FUNCTION_BLOCK Path1d EXTENDS ZCore.Object IMPLEMENTS IPathQuery, IPathQuery2, IPathQuery3, ZCore.IUnmanagedObject
VAR
  _owner : REFERENCE TO Unit;
  _fromPosition, _toPosition : LREAL;
  _direction : INT;
  _halfWidth, _safetyMargin : LREAL;
  _regions : POINTER TO ZApplication.IRegion;
  _regionEnd : INT;
  
  _maxRegions : DINT := 5;
  _regionIndicesBuffer1 : ARRAY[0..5] OF INT;
  _regionIndicesBuffer2 : ARRAY[0..5] OF INT;  
  _regionLockIndices : ZCore.RingBufferInt(_maxRegions, ADR(_regionIndicesBuffer1));
  _regionUnlockIndices : ZCore.RingBufferInt(_maxRegions, ADR(_regionIndicesBuffer2));
END_VAR

METHOD CheckAndLock : BOOL;
VAR_INPUT
  pos : LREAL;
END_VAR
VAR_INST
  i : DINT;
  region : ZApplication.IRegion;
  corner1WithMargin, corner2WithMargin : Vector4;
END_VAR
IF _regionLockIndices.Empty
THEN
  CheckAndLock := TRUE;
  RETURN;
END_IF

region := _regions[_regionLockIndices.ItemAt(0)];
CheckAndLock := 
  region.IntersectsIntervalX(pos - _halfWidth - _safetyMargin, pos + _halfWidth + _safetyMargin) AND_THEN
  region.TryLock(_owner);
  
IF CheckAndLock
THEN
  _regionUnlockIndices.Append(_regionLockIndices.ItemAt(0));
END_IF
END_METHOD

PROPERTY CurrentEdge : LREAL
GET
IF _regionLockIndices.Empty
THEN
  CurrentEdge := _toPosition;
  RETURN;
END_IF

IF _direction < 0
THEN
  CurrentEdge := _regions[_regionLockIndices.ItemAt(0)].Corner2.X + _halfWidth;
ELSE
  CurrentEdge := _regions[_regionLockIndices.ItemAt(0)].Corner1.X - _halfWidth;
END_IF
END_GET
END_PROPERTY

METHOD Cyclic
VAR_INST
  i : DINT;
  region : ZApplication.IRegion;
  priority : INT;
  priorityIndex : DINT;
  waiting : BOOL;
END_VAR
IF NOT Busy
THEN
  RETURN;
END_IF

IF _regionLockIndices.Empty
THEN
  SetBusy(FALSE);  
  RETURN;
END_IF

priority := 10000;
FOR i := 0 TO _regionLockIndices.Size - 1
DO
  region := _regions[_regionLockIndices.ItemAt(i)];
  IF priority > region.Priority
  THEN
    priorityIndex := i;
    priority := region.Priority;
  END_IF
END_FOR

waiting := FALSE;
FOR i := priorityIndex TO _regionLockIndices.Size - 1
DO
  region := _regions[_regionLockIndices.ItemAt(i)];
  IF NOT region.TryLock(_owner)
  THEN
    waiting := TRUE;
  END_IF
END_FOR

SetBusy(waiting);

// We can't move so free up resources
IF Busy
THEN
  FOR i := 0 TO _regionLockIndices.Size - 1
  DO
    region := _regions[_regionLockIndices.ItemAt(i)];
    region.Unlock(_owner);
  END_FOR
END_IF
END_METHOD

//FB_Init is always available implicitly and it is used primarily for initialization.
//The return value is not evaluated. For a specific influence, you can also declare the
//methods explicitly and provide additional code there with the standard initialization
//code. You can evaluate the return value.
METHOD FB_Init: BOOL
VAR_INPUT
    bInitRetains: BOOL; // TRUE: the retain variables are initialized (reset warm / reset cold)
    bInCopyCode: BOOL;  // TRUE: the instance will be copied to the copy code afterward (online change)   
END_VAR
SetIdle();
END_METHOD

METHOD FromPosition : IPathQuery2
VAR_INPUT
  pos : LREAL;
END_VAR
_fromPosition := pos;

FromPosition := THIS^;
END_METHOD

METHOD IncrementRegion
VAR_INST
  intervalMin : LREAL;
  intervalMax : LREAL;
  i : INT;
  
  corner1, corner2 : Vector4;
END_VAR
IF NOT _regionLockIndices.Empty
THEN
  _regionLockIndices.PopFirstItem();
END_IF
END_METHOD

PROPERTY RegionsToPass : DINT
GET
RegionsToPass := _regionLockIndices.Size;
END_GET
END_PROPERTY

METHOD ReserveAsync
VAR_INPUT
  unit : REFERENCE TO Unit;
END_VAR
VAR_INST
  intervalMin : LREAL;
  intervalMax : LREAL;
  i, start, end : INT;
END_VAR
intervalMin := MIN(_fromPosition - _halfWidth, _toPosition - _halfWidth);
intervalMax := MAX(_fromPosition + _halfWidth, _toPosition + _halfWidth);

_owner REF= unit;
_direction := SEL(_fromPosition < _toPosition, -1, 1);

_regionLockIndices.Clear();
_regionUnlockIndices.Clear();

IF _direction < 0
THEN
  start := _regionEnd;
  end := 0;
ELSE
  start := 0;
  end := _regionEnd;
END_IF

FOR i := start TO end BY _direction
DO
  IF _regions[i].IntersectsIntervalX(intervalMin, intervalMax)
  THEN
    _regionLockIndices.Append(i);
  END_IF
END_FOR

SetBusy(TRUE);
END_METHOD

METHOD ToPosition : IPathQuery3
VAR_INPUT
  pos : LREAL;
END_VAR
_toPosition := pos;

ToPosition := THIS^;
END_METHOD

METHOD UnlockPassedRegions : IError
VAR_INPUT
  pos : LREAL;
END_VAR
VAR_INST
  i : DINT;
  region : ZApplication.IRegion;
END_VAR
IF NOT _regionUnlockIndices.Empty
THEN
  region := _regions[_regionUnlockIndices.ItemAt(0)];
  WHILE (_direction < 0 AND_THEN pos + _halfWidth < region.Corner1.X) OR_ELSE
        (_direction > 0 AND_THEN pos - _halfWidth > region.Corner2.X)
  DO
    region.Unlock(_owner);
    _regionUnlockIndices.PopFirstItem();
    
    IF _regionUnlockIndices.Empty
    THEN
      EXIT;
    END_IF
    
    region := _regions[_regionUnlockIndices.ItemAt(0)];
  END_WHILE
END_IF
END_METHOD

METHOD WithSafetyMargin : IPathQuery
VAR_INPUT
  margin : LREAL;
END_VAR
_safetyMargin := margin;

WithSafetyMargin := THIS^;
END_METHOD

METHOD WithSortedRegions : IPathQuery
VAR_INPUT
  regions : POINTER TO ZApplication.IRegion;
  regionCount : INT;
END_VAR
_regions := regions;
_regionEnd := regionCount-1;

WithSortedRegions := THIS^;
END_METHOD

METHOD WithWidth : IPathQuery
VAR_INPUT
  width : LREAL;
END_VAR
_halfWidth := width * 0.5;

WithWidth := THIS^;
END_METHOD

END_FUNCTION_BLOCK

(* stored: Version 1.1.0.1
   POU Path1d: Id {d163563b-b0d8-0bc3-395b-6d8352dd5158}, SpecialFunc None
   Method CheckAndLock: Id {d0ea5090-f040-4e8b-b4d9-204aa228834b}
   Property CurrentEdge: Id {4c10ff27-4f30-4d44-a9f9-0de27afcd8bd}
   Get Get: Id {bed5760d-ad6a-434f-bc42-ef8e41897a33}
   Method Cyclic: Id {2f8e18f1-7b9f-43ca-9807-35cbe99480a6}
   Method FB_Init: Id {b6ede0be-ab8f-47f6-bb7f-2b9119232049}
   Method FromPosition: Id {c717db84-1e2a-0be7-378a-a2d2a7d60e6a}
   Method IncrementRegion: Id {39e24ae9-687e-4ea8-bac4-6000ef29c62e}
   Property RegionsToPass: Id {79686e52-b356-4ca7-a824-1164c5bff563}
   Get Get: Id {747df01b-e3d2-4965-affb-874dc140a240}
   Method ReserveAsync: Id {e607f347-fe2e-07c1-1baf-c06f8dc6270a}
   Method ToPosition: Id {96a0486b-dd4f-0cad-3260-b33f67f5e78b}
   Method UnlockPassedRegions: Id {ce34f11a-e22e-422e-8b3c-8bccb88f81dd}
   Method WithSafetyMargin: Id {652e493c-1f38-430b-962f-8a16e35509de}
   Method WithSortedRegions: Id {d968df69-3240-4dd9-ab3d-cb58fae1f925}
   Method WithWidth: Id {b0e59529-3f47-4d26-bdcf-c3f5c7e23a81} *)
